FUNCTION_BLOCK IN_ENUM_CTL (* Control block for IN_ENUM *)
  (* Standard: 61499-2 *)
  (* Version 0.1, 2006-04-21, JHC, Holobloc Inc, Added service sequences *)
  (* Version 0.0, 2004-06-21, JHC, Rockwell Automation *)
  (* Compiler header: package fb.rt.hmi; *)
  (* Compiler Java Sun JDK 1.5.0 *)
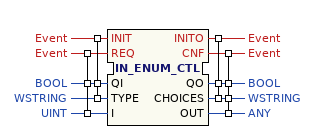
  EVENT_INPUT
    INIT WITH QI, TYPE; (* Service Initialization *)
    REQ WITH QI, I; (* Service Request *)
  END_EVENT
  EVENT_OUTPUT
    INITO WITH QO, CHOICES; (* Initialization Confirm *)
    CNF WITH QO, CHOICES, OUT; (* Confirmation of Requested Service *)
  END_EVENT
  VAR_INPUT
    QI : BOOL; (* Event Input Qualifier *)
    TYPE : WSTRING; (* Enumerated Type Name *)
    I : UINT; (* Current enumerated index *)
  END_VAR
  VAR_OUTPUT
    QO : BOOL; (* Event Output Qualifier *)
    CHOICES : WSTRING; (* Comma-separated enumeration namelist *)
    OUT : ANY; (* Enumerated variable with selected value *)
  END_VAR
  SERVICE APPLICATION/RESOURCE
    SEQUENCE initialize
      APPLICATION.INIT+(TYPE) -> RESOURCE.checkType(TYPE) -> RESOURCE.getChoices(TYPE) -> APPLICATION.INITO+(CHOICES);
    END_SEQUENCE
    SEQUENCE invalid_type
      APPLICATION.INIT+(TYPE) -> RESOURCE.checkType(TYPE) -> RESOURCE.removeAllChoices() -> APPLICATION.INITO-(CHOICES);
    END_SEQUENCE
    SEQUENCE select
      APPLICATION.REQ+(I) -> RESOURCE.getChoice(I) -> APPLICATION.CNF+(OUT);
    END_SEQUENCE
    SEQUENCE select_inhibited
      APPLICATION.REQ-() -> APPLICATION.CNF-();
    END_SEQUENCE
    SEQUENCE terminate
      APPLICATION.INIT-() -> RESOURCE.removeAllChoices() -> APPLICATION.INITO-(CHOICES);
    END_SEQUENCE
  END_SERVICE
END_FUNCTION_BLOCK
